Universal Robots PolyScope program: smrttt_with_blends_online.urp

Program smrttt_with_blends_online (installation=default directory=/programs createdIn=5.14.5 lastSavedIn=5.14.5 robotSerialNumber=20236801216)
Calibrated DH parameters: a=[-0.000021, -0.748897, -0.28186, -0.00004, -0.000055, 0]; d=[0.236225, -424.082933, -1564.66872, 1988.95162, 0.159094, 0.153873]; alpha=[1.570844, 0.001002, 0.000337, 1.571488, -1.569996, 0]; deltaTheta=[0, -0.516316, 5.626292, 1.173211, 0.000001, 0]
InitVariablesNode
Robot Program (runOnlyOnce=false)
  start_pos := get_forward_kin()
  height :=  (valueSource=Operator message=Height in mm? valueType=Float)
  width :=  (valueSource=Operator message=Width in mm? valueType=Float)
  Loop Forever
    MoveL speed 250 mm/s, acceleration 1200 mm/s^2 (useActiveTCP=true) feature=Base
      corner_1 := pose_trans(start_pos,p[width/1000.0,0.0,0.0,0.0,0.0,0.0])
      Waypoint Variable (Variable): variable=corner_1
    MoveL speed 250 mm/s, acceleration 1200 mm/s^2 (useActiveTCP=true) feature=Base
      corner_2 := pose_trans(start_pos,p[width/1000.0,height/1000.0,0.0,0.0,0.0,0.0])
      Waypoint Variable (Variable): variable=corner_2
    MoveL speed 250 mm/s, acceleration 1200 mm/s^2 (useActiveTCP=true) feature=Base
      corner_3 := pose_trans(start_pos,p[0.0,height/1000.0,0.0,0.0,0.0,0.0])
      Waypoint Variable (Variable): variable=corner_3
    MoveL speed 250 mm/s, acceleration 1200 mm/s^2 (useActiveTCP=true) feature=Base
      Waypoint Variable (Variable): variable=start_pos
